PROGRAM ReelCommand
VAR
	Zero: MC_SetPosition;
	power: MC_Power;
	MC_MoveAbsolute: MC_MoveAbsolute;
	MC_Jog_0: MC_Jog;
	FB_CoEAX8000BrakeControl_0: FB_CoEAX8000BrakeControl;
	Release: BOOL;
	Brake: E_BrakeMode := eBrakeMode_Unlock;
	VeloLeading: MC_MoveAbsolute;
	bVeloStart: BOOL;
	R_TRIG_0: R_TRIG;
	
	Cutout			:bool;
	
	velolatch		at %I* : BOOL;
	F_trig_0: f_TRIG;
	MC_MoveAbsolute_ForJeff: MC_MoveAbsolute;
END_VAR

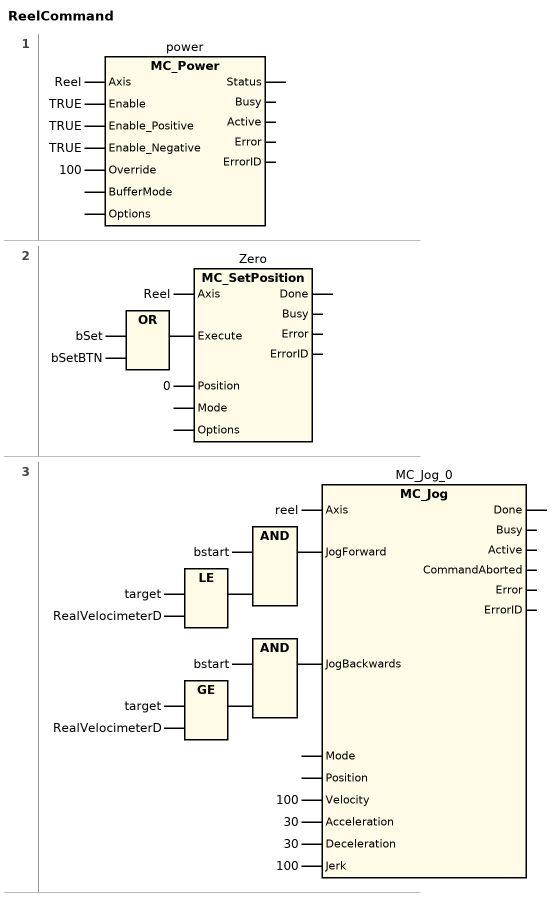
// NETWORK 1
power(Axis := Reel, Enable := TRUE, Enable_Positive := TRUE, Enable_Negative := TRUE, Override := 100); // MC_Power

// NETWORK 2
Zero(Axis := Reel, Execute := bSet OR bSetBTN, Position := 0); // MC_SetPosition

// NETWORK 3
MC_Jog_0(
    Axis := reel,
    JogForward := bstart AND target <= RealVelocimeterD,
    JogBackwards := bstart AND target >= RealVelocimeterD,
    Velocity := 100,
    Acceleration := 30,
    Deceleration := 30,
    Jerk := 100); // MC_Jog

END_PROGRAM

(* stored: Version 1.1.0.1, ProductVersion 3.1.4024.12
   POU ReelCommand: Id {d557e279-5996-4de8-b528-0b9d0286dce8}, SpecialFunc None *)
